FUNCTION_BLOCK fbToleranceTimeCtrl
VAR_INPUT

	bEnable					: BOOL;
	bBasketCFM				: BOOL;
	bProcessCompleted		: BOOL;
	iToleranceTimeSv		: INT;


END_VAR
VAR_OUTPUT

	bAssignBadBstBit		: BOOL;
	iToleranceTimePV	: INT;

END_VAR
VAR
	TON1: TON;
	TON2: TON;
	bAssignBadBstBitInt: BOOL;
END_VAR
VAR // added by the converter: edge detectors and wires of the graphical bodies
    _w1 : ANY;
    _w2 : INT;
END_VAR

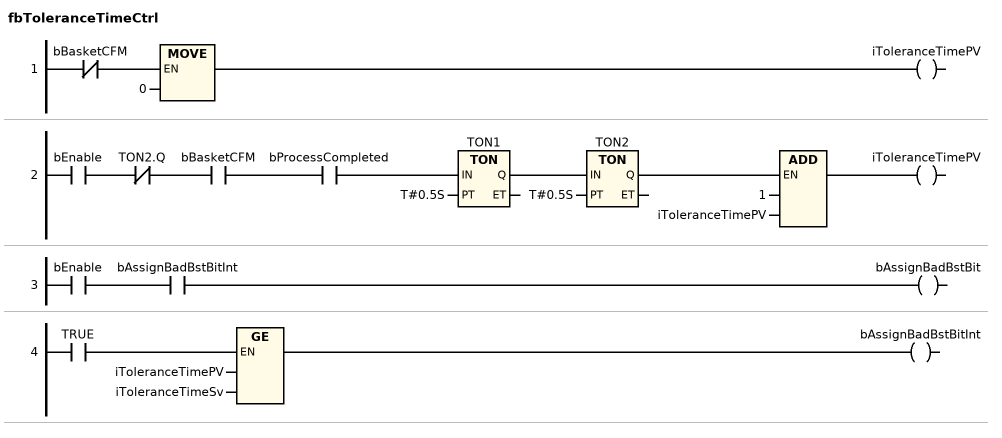
// NETWORK 1
IF NOT bBasketCFM THEN _w1 := 0; END_IF
iToleranceTimePV := _w1;

// NETWORK 2
TON1(IN := bEnable AND NOT TON2.Q AND bBasketCFM AND bProcessCompleted, PT := T#0.5S); // TON
TON2(IN := TON1.Q, PT := T#0.5S); // TON
IF TON2.Q THEN _w2 := 1 + iToleranceTimePV; END_IF
iToleranceTimePV := _w2;

// NETWORK 3
bAssignBadBstBit := bEnable AND bAssignBadBstBitInt;

// NETWORK 4
bAssignBadBstBitInt := iToleranceTimePV >= iToleranceTimeSv;

END_FUNCTION_BLOCK

(* stored: Version 1.1.0.1, ProductVersion 3.1.4024.12
   POU fbToleranceTimeCtrl: Id {232f8287-27ef-44cb-994d-3dd12b15bf6d}, SpecialFunc None *)
